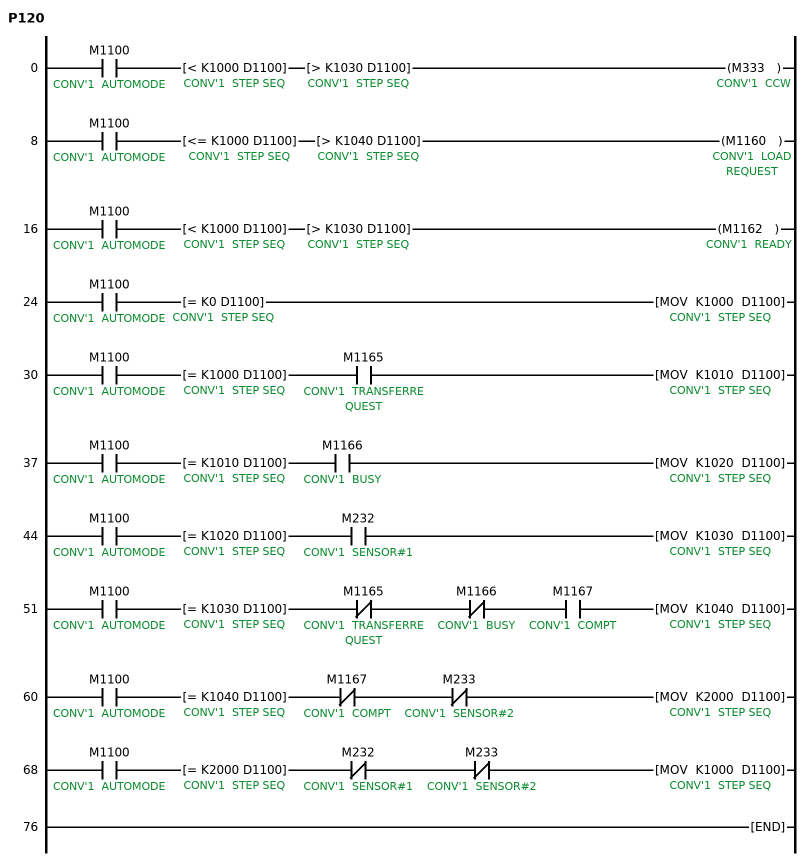
[picture p24: ladder of P120, rungs at steps 0 to 76]
0     LD      M1100  ; CONV'1  AUTOMODE
      AND<    K1000 D1100  ; CONV'1  STEP SEQ
      AND>    K1030 D1100  ; CONV'1  STEP SEQ
      OUT     M333  ; CONV'1  CCW
8     LD      M1100  ; CONV'1  AUTOMODE
      AND<=   K1000 D1100  ; CONV'1  STEP SEQ
      AND>    K1040 D1100  ; CONV'1  STEP SEQ
      OUT     M1160  ; CONV'1  LOAD    REQUEST
16    LD      M1100  ; CONV'1  AUTOMODE
      AND<    K1000 D1100  ; CONV'1  STEP SEQ
      AND>    K1030 D1100  ; CONV'1  STEP SEQ
      OUT     M1162  ; CONV'1  READY
24    LD      M1100  ; CONV'1  AUTOMODE
      AND=    K0 D1100  ; CONV'1  STEP SEQ
      MOV     K1000 D1100
30    LD      M1100  ; CONV'1  AUTOMODE
      AND=    K1000 D1100  ; CONV'1  STEP SEQ
      AND     M1165  ; CONV'1  TRANSFERREQUEST
      MOV     K1010 D1100
37    LD      M1100  ; CONV'1  AUTOMODE
      AND=    K1010 D1100  ; CONV'1  STEP SEQ
      AND     M1166  ; CONV'1  BUSY
      MOV     K1020 D1100
44    LD      M1100  ; CONV'1  AUTOMODE
      AND=    K1020 D1100  ; CONV'1  STEP SEQ
      AND     M232  ; CONV'1  SENSOR#1
      MOV     K1030 D1100
51    LD      M1100  ; CONV'1  AUTOMODE
      AND=    K1030 D1100  ; CONV'1  STEP SEQ
      ANI     M1165  ; CONV'1  TRANSFERREQUEST
      ANI     M1166  ; CONV'1  BUSY
      AND     M1167  ; CONV'1  COMPT
      MOV     K1040 D1100
60    LD      M1100  ; CONV'1  AUTOMODE
      AND=    K1040 D1100  ; CONV'1  STEP SEQ
      ANI     M1167  ; CONV'1  COMPT
      ANI     M233  ; CONV'1  SENSOR#2
      MOV     K2000 D1100
68    LD      M1100  ; CONV'1  AUTOMODE
      AND=    K2000 D1100  ; CONV'1  STEP SEQ
      ANI     M232  ; CONV'1  SENSOR#1
      ANI     M233  ; CONV'1  SENSOR#2
      MOV     K1000 D1100
76    END
END_PROGRAM

PROGRAM P130  // CONV2
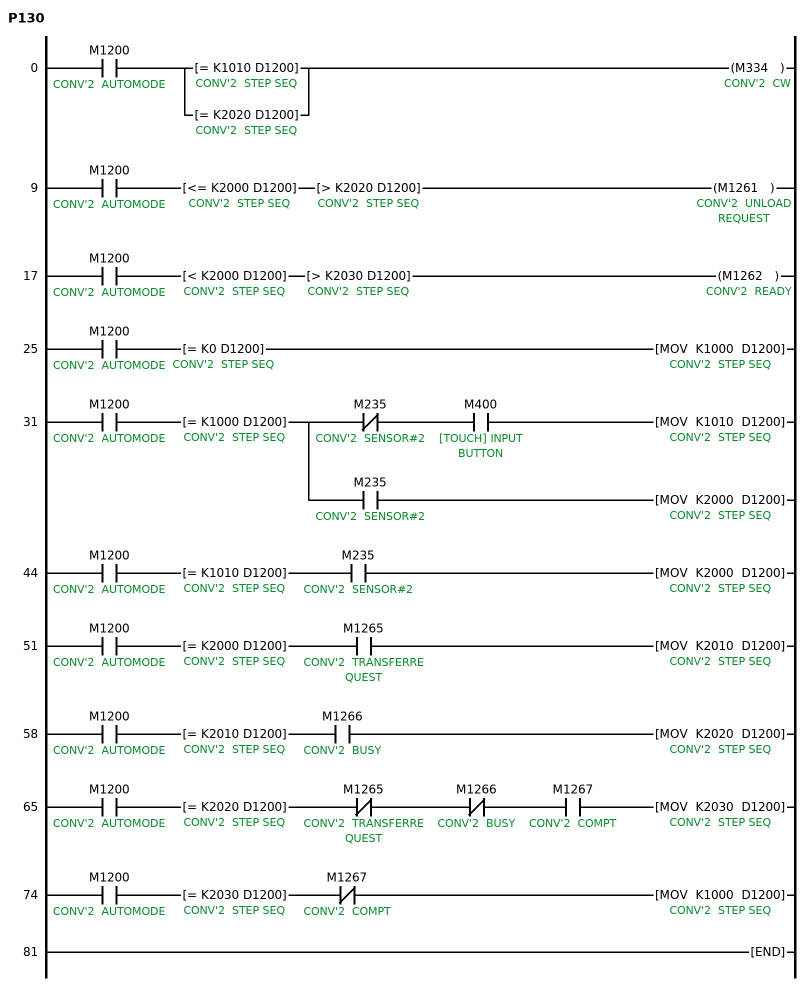
0     LD      M1200  ; CONV'2  AUTOMODE
      LD=     K1010 D1200  ; CONV'2  STEP SEQ
      OR=     K2020 D1200  ; CONV'2  STEP SEQ
      ANB
      OUT     M334  ; CONV'2  CW
9     LD      M1200  ; CONV'2  AUTOMODE
      AND<=   K2000 D1200  ; CONV'2  STEP SEQ
      AND>    K2020 D1200  ; CONV'2  STEP SEQ
      OUT     M1261  ; CONV'2  UNLOAD  REQUEST
17    LD      M1200  ; CONV'2  AUTOMODE
      AND<    K2000 D1200  ; CONV'2  STEP SEQ
      AND>    K2030 D1200  ; CONV'2  STEP SEQ
      OUT     M1262  ; CONV'2  READY
25    LD      M1200  ; CONV'2  AUTOMODE
      AND=    K0 D1200  ; CONV'2  STEP SEQ
      MOV     K1000 D1200
31    LD      M1200  ; CONV'2  AUTOMODE
      AND=    K1000 D1200  ; CONV'2  STEP SEQ
      MPS
      ANI     M235  ; CONV'2  SENSOR#2
      AND     M400  ; [TOUCH] INPUT   BUTTON
      MOV     K1010 D1200
      MPP
      AND     M235  ; CONV'2  SENSOR#2
      MOV     K2000 D1200
44    LD      M1200  ; CONV'2  AUTOMODE
      AND=    K1010 D1200  ; CONV'2  STEP SEQ
      AND     M235  ; CONV'2  SENSOR#2
      MOV     K2000 D1200
51    LD      M1200  ; CONV'2  AUTOMODE
      AND=    K2000 D1200  ; CONV'2  STEP SEQ
      AND     M1265  ; CONV'2  TRANSFERREQUEST
      MOV     K2010 D1200
58    LD      M1200  ; CONV'2  AUTOMODE
      AND=    K2010 D1200  ; CONV'2  STEP SEQ
      AND     M1266  ; CONV'2  BUSY
      MOV     K2020 D1200
65    LD      M1200  ; CONV'2  AUTOMODE
      AND=    K2020 D1200  ; CONV'2  STEP SEQ
      ANI     M1265  ; CONV'2  TRANSFERREQUEST
      ANI     M1266  ; CONV'2  BUSY
      AND     M1267  ; CONV'2  COMPT
      MOV     K2030 D1200
74    LD      M1200  ; CONV'2  AUTOMODE
      AND=    K2030 D1200  ; CONV'2  STEP SEQ
      ANI     M1267  ; CONV'2  COMPT
      MOV     K1000 D1200
81    END
END_PROGRAM

PROGRAM P140  // CONV3
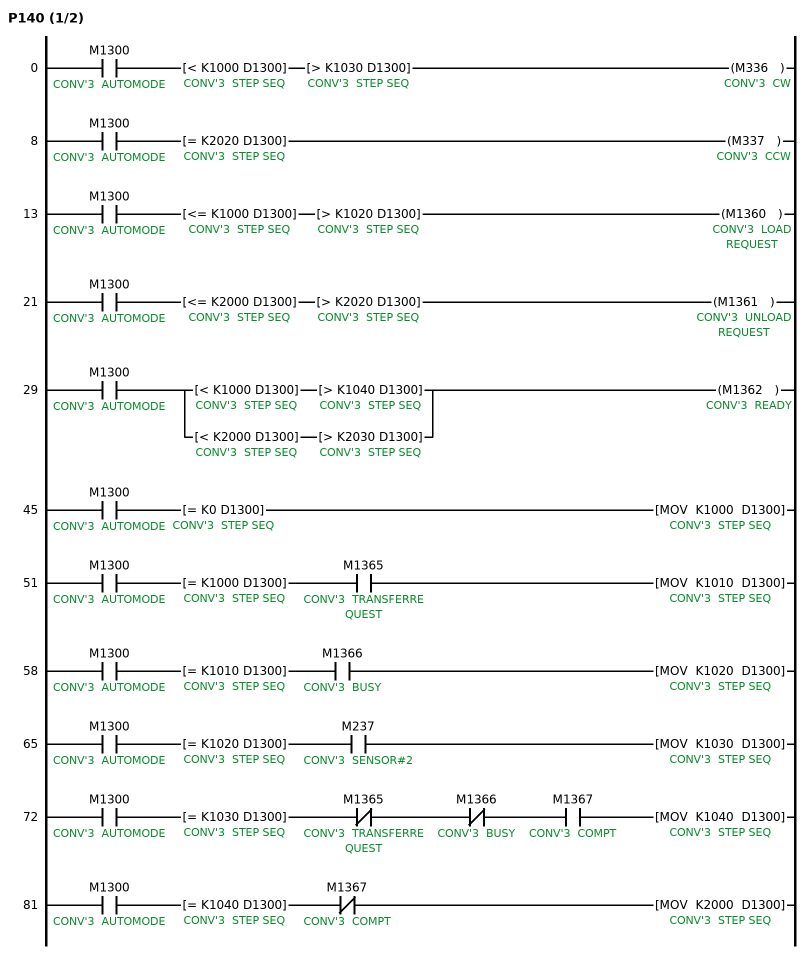
0     LD      M1300  ; CONV'3  AUTOMODE
      AND<    K1000 D1300  ; CONV'3  STEP SEQ
      AND>    K1030 D1300  ; CONV'3  STEP SEQ
      OUT     M336  ; CONV'3  CW
8     LD      M1300  ; CONV'3  AUTOMODE
      AND=    K2020 D1300  ; CONV'3  STEP SEQ
      OUT     M337  ; CONV'3  CCW
13    LD      M1300  ; CONV'3  AUTOMODE
      AND<=   K1000 D1300  ; CONV'3  STEP SEQ
      AND>    K1020 D1300  ; CONV'3  STEP SEQ
      OUT     M1360  ; CONV'3  LOAD    REQUEST
21    LD      M1300  ; CONV'3  AUTOMODE
      AND<=   K2000 D1300  ; CONV'3  STEP SEQ
      AND>    K2020 D1300  ; CONV'3  STEP SEQ
      OUT     M1361  ; CONV'3  UNLOAD  REQUEST
29    LD      M1300  ; CONV'3  AUTOMODE
      LD<     K1000 D1300  ; CONV'3  STEP SEQ
      AND>    K1040 D1300  ; CONV'3  STEP SEQ
      LD<     K2000 D1300  ; CONV'3  STEP SEQ
      AND>    K2030 D1300  ; CONV'3  STEP SEQ
      ORB
      ANB
      OUT     M1362  ; CONV'3  READY
45    LD      M1300  ; CONV'3  AUTOMODE
      AND=    K0 D1300  ; CONV'3  STEP SEQ
      MOV     K1000 D1300
51    LD      M1300  ; CONV'3  AUTOMODE
      AND=    K1000 D1300  ; CONV'3  STEP SEQ
      AND     M1365  ; CONV'3  TRANSFERREQUEST
      MOV     K1010 D1300
58    LD      M1300  ; CONV'3  AUTOMODE
      AND=    K1010 D1300  ; CONV'3  STEP SEQ
      AND     M1366  ; CONV'3  BUSY
      MOV     K1020 D1300
65    LD      M1300  ; CONV'3  AUTOMODE
      AND=    K1020 D1300  ; CONV'3  STEP SEQ
      AND     M237  ; CONV'3  SENSOR#2
      MOV     K1030 D1300
72    LD      M1300  ; CONV'3  AUTOMODE
      AND=    K1030 D1300  ; CONV'3  STEP SEQ
      ANI     M1365  ; CONV'3  TRANSFERREQUEST
      ANI     M1366  ; CONV'3  BUSY
      AND     M1367  ; CONV'3  COMPT
      MOV     K1040 D1300
81    LD      M1300  ; CONV'3  AUTOMODE
      AND=    K1040 D1300  ; CONV'3  STEP SEQ
      ANI     M1367  ; CONV'3  COMPT
      MOV     K2000 D1300
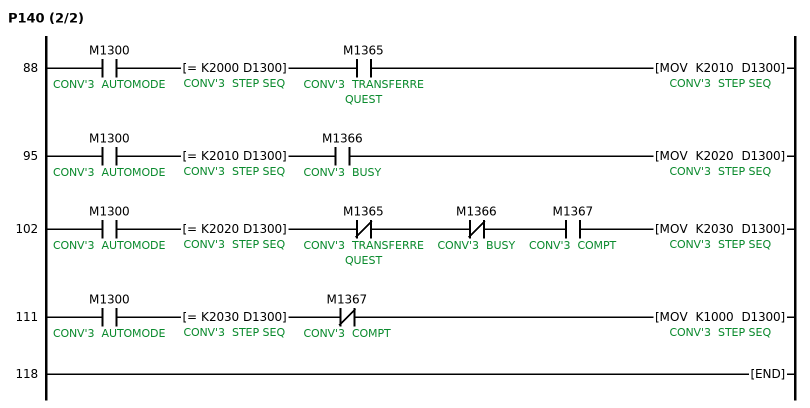
88    LD      M1300  ; CONV'3  AUTOMODE
      AND=    K2000 D1300  ; CONV'3  STEP SEQ
      AND     M1365  ; CONV'3  TRANSFERREQUEST
      MOV     K2010 D1300
95    LD      M1300  ; CONV'3  AUTOMODE
      AND=    K2010 D1300  ; CONV'3  STEP SEQ
      AND     M1366  ; CONV'3  BUSY
      MOV     K2020 D1300
102   LD      M1300  ; CONV'3  AUTOMODE
      AND=    K2020 D1300  ; CONV'3  STEP SEQ
      ANI     M1365  ; CONV'3  TRANSFERREQUEST
      ANI     M1366  ; CONV'3  BUSY
      AND     M1367  ; CONV'3  COMPT
      MOV     K2030 D1300
111   LD      M1300  ; CONV'3  AUTOMODE
      AND=    K2030 D1300  ; CONV'3  STEP SEQ
      ANI     M1367  ; CONV'3  COMPT
      MOV     K1000 D1300
118   END
END_PROGRAM

PROGRAM P150  // CONV4
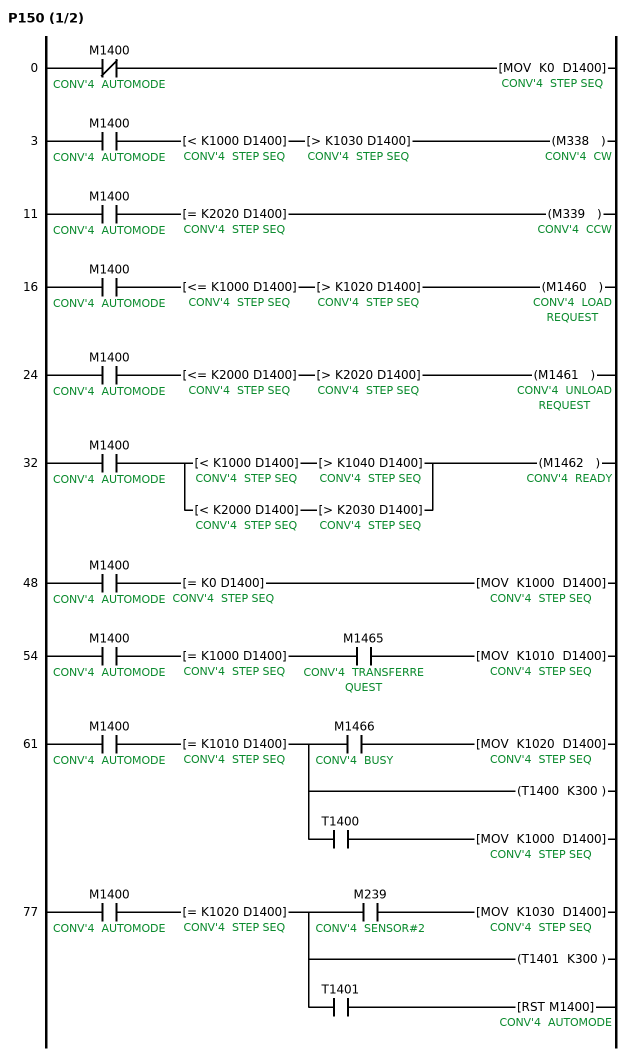
0     LDI     M1400  ; CONV'4  AUTOMODE
      MOV     K0 D1400  ; CONV'4  STEP SEQ
3     LD      M1400  ; CONV'4  AUTOMODE
      AND<    K1000 D1400  ; CONV'4  STEP SEQ
      AND>    K1030 D1400  ; CONV'4  STEP SEQ
      OUT     M338  ; CONV'4  CW
11    LD      M1400  ; CONV'4  AUTOMODE
      AND=    K2020 D1400  ; CONV'4  STEP SEQ
      OUT     M339  ; CONV'4  CCW
16    LD      M1400  ; CONV'4  AUTOMODE
      AND<=   K1000 D1400  ; CONV'4  STEP SEQ
      AND>    K1020 D1400  ; CONV'4  STEP SEQ
      OUT     M1460  ; CONV'4  LOAD    REQUEST
24    LD      M1400  ; CONV'4  AUTOMODE
      AND<=   K2000 D1400  ; CONV'4  STEP SEQ
      AND>    K2020 D1400  ; CONV'4  STEP SEQ
      OUT     M1461  ; CONV'4  UNLOAD  REQUEST
32    LD      M1400  ; CONV'4  AUTOMODE
      LD<     K1000 D1400  ; CONV'4  STEP SEQ
      AND>    K1040 D1400  ; CONV'4  STEP SEQ
      LD<     K2000 D1400  ; CONV'4  STEP SEQ
      AND>    K2030 D1400  ; CONV'4  STEP SEQ
      ORB
      ANB
      OUT     M1462  ; CONV'4  READY
48    LD      M1400  ; CONV'4  AUTOMODE
      AND=    K0 D1400  ; CONV'4  STEP SEQ
      MOV     K1000 D1400
54    LD      M1400  ; CONV'4  AUTOMODE
      AND=    K1000 D1400  ; CONV'4  STEP SEQ
      AND     M1465  ; CONV'4  TRANSFERREQUEST
      MOV     K1010 D1400
61    LD      M1400  ; CONV'4  AUTOMODE
      AND=    K1010 D1400  ; CONV'4  STEP SEQ
      MPS
      AND     M1466  ; CONV'4  BUSY
      MOV     K1020 D1400
      MPP
      OUT     T1400 K300
      AND     T1400
      MOV     K1000 D1400
77    LD      M1400  ; CONV'4  AUTOMODE
      AND=    K1020 D1400  ; CONV'4  STEP SEQ
      MPS
      AND     M239  ; CONV'4  SENSOR#2
      MOV     K1030 D1400
      MPP
      OUT     T1401 K300
      AND     T1401
      RST     M1400  ; CONV'4  AUTOMODE
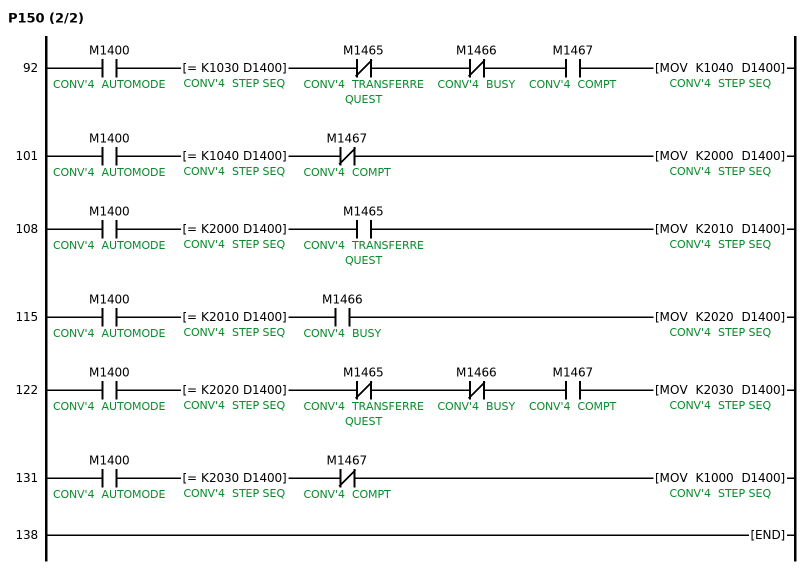
92    LD      M1400  ; CONV'4  AUTOMODE
      AND=    K1030 D1400  ; CONV'4  STEP SEQ
      ANI     M1465  ; CONV'4  TRANSFERREQUEST
      ANI     M1466  ; CONV'4  BUSY
      AND     M1467  ; CONV'4  COMPT
      MOV     K1040 D1400
101   LD      M1400  ; CONV'4  AUTOMODE
      AND=    K1040 D1400  ; CONV'4  STEP SEQ
      ANI     M1467  ; CONV'4  COMPT
      MOV     K2000 D1400
108   LD      M1400  ; CONV'4  AUTOMODE
      AND=    K2000 D1400  ; CONV'4  STEP SEQ
      AND     M1465  ; CONV'4  TRANSFERREQUEST
      MOV     K2010 D1400
115   LD      M1400  ; CONV'4  AUTOMODE
      AND=    K2010 D1400  ; CONV'4  STEP SEQ
      AND     M1466  ; CONV'4  BUSY
      MOV     K2020 D1400
122   LD      M1400  ; CONV'4  AUTOMODE
      AND=    K2020 D1400  ; CONV'4  STEP SEQ
      ANI     M1465  ; CONV'4  TRANSFERREQUEST
      ANI     M1466  ; CONV'4  BUSY
      AND     M1467  ; CONV'4  COMPT
      MOV     K2030 D1400
131   LD      M1400  ; CONV'4  AUTOMODE
      AND=    K2030 D1400  ; CONV'4  STEP SEQ
      ANI     M1467  ; CONV'4  COMPT
      MOV     K1000 D1400
138   END
END_PROGRAM

PROGRAM P100  // MODE
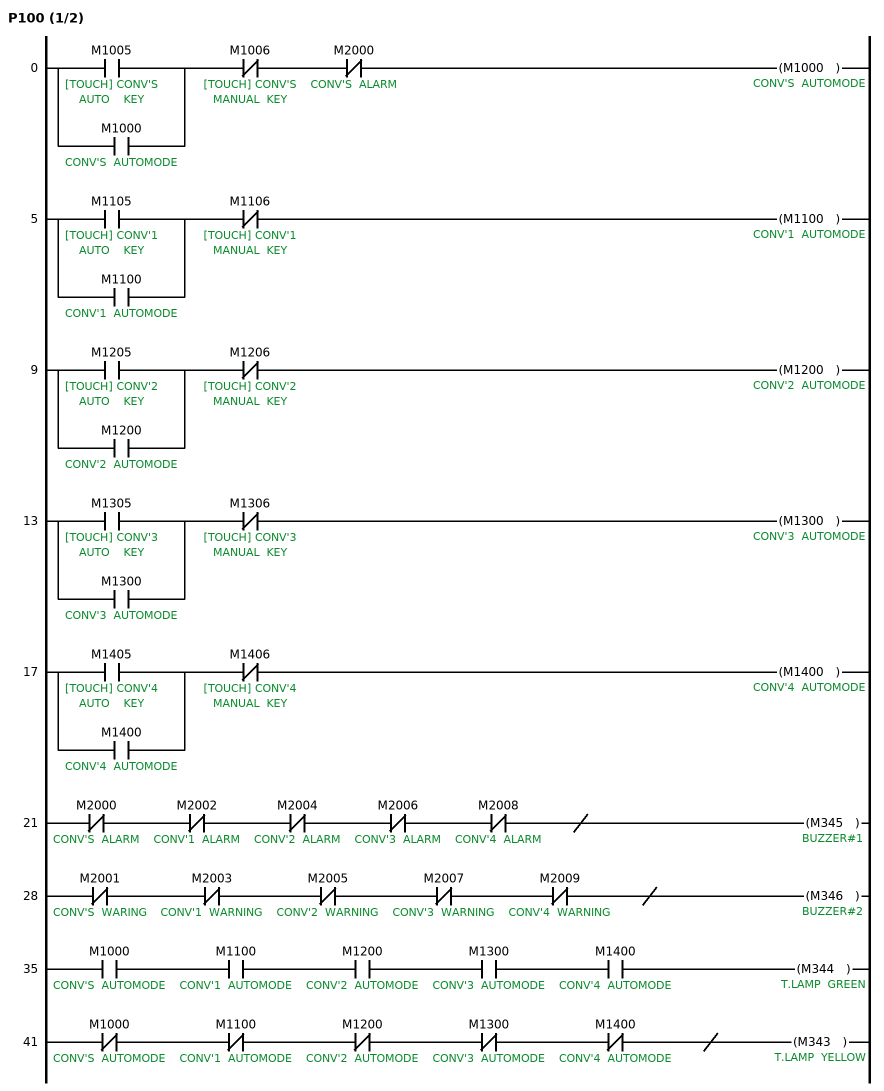
0     LD      M1005  ; [TOUCH] CONV'S  AUTO    KEY
      OR      M1000  ; CONV'S  AUTOMODE
      ANI     M1006  ; [TOUCH] CONV'S  MANUAL  KEY
      ANI     M2000  ; CONV'S  ALARM
      OUT     M1000  ; CONV'S  AUTOMODE
5     LD      M1105  ; [TOUCH] CONV'1  AUTO    KEY
      OR      M1100  ; CONV'1  AUTOMODE
      ANI     M1106  ; [TOUCH] CONV'1  MANUAL  KEY
      OUT     M1100  ; CONV'1  AUTOMODE
9     LD      M1205  ; [TOUCH] CONV'2  AUTO    KEY
      OR      M1200  ; CONV'2  AUTOMODE
      ANI     M1206  ; [TOUCH] CONV'2  MANUAL  KEY
      OUT     M1200  ; CONV'2  AUTOMODE
13    LD      M1305  ; [TOUCH] CONV'3  AUTO    KEY
      OR      M1300  ; CONV'3  AUTOMODE
      ANI     M1306  ; [TOUCH] CONV'3  MANUAL  KEY
      OUT     M1300  ; CONV'3  AUTOMODE
17    LD      M1405  ; [TOUCH] CONV'4  AUTO    KEY
      OR      M1400  ; CONV'4  AUTOMODE
      ANI     M1406  ; [TOUCH] CONV'4  MANUAL  KEY
      OUT     M1400  ; CONV'4  AUTOMODE
21    LDI     M2000  ; CONV'S  ALARM
      ANI     M2002  ; CONV'1  ALARM
      ANI     M2004  ; CONV'2  ALARM
      ANI     M2006  ; CONV'3  ALARM
      ANI     M2008  ; CONV'4  ALARM
      INV
      OUT     M345  ; BUZZER#1
28    LDI     M2001  ; CONV'S  WARING
      ANI     M2003  ; CONV'1  WARNING
      ANI     M2005  ; CONV'2  WARNING
      ANI     M2007  ; CONV'3  WARNING
      ANI     M2009  ; CONV'4  WARNING
      INV
      OUT     M346  ; BUZZER#2
35    LD      M1000  ; CONV'S  AUTOMODE
      AND     M1100  ; CONV'1  AUTOMODE
      AND     M1200  ; CONV'2  AUTOMODE
      AND     M1300  ; CONV'3  AUTOMODE
      AND     M1400  ; CONV'4  AUTOMODE
      OUT     M344  ; T.LAMP  GREEN
41    LDI     M1000  ; CONV'S  AUTOMODE
      ANI     M1100  ; CONV'1  AUTOMODE
      ANI     M1200  ; CONV'2  AUTOMODE
      ANI     M1300  ; CONV'3  AUTOMODE
      ANI     M1400  ; CONV'4  AUTOMODE
      INV
      OUT     M343  ; T.LAMP  YELLOW
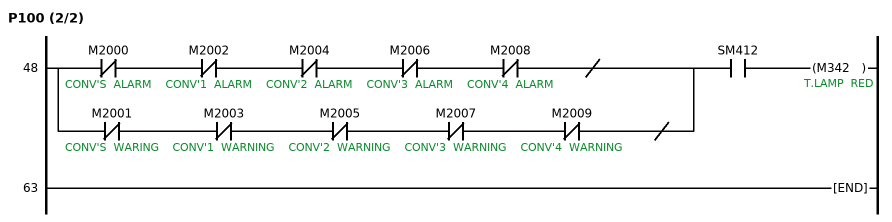
48    LDI     M2000  ; CONV'S  ALARM
      ANI     M2002  ; CONV'1  ALARM
      ANI     M2004  ; CONV'2  ALARM
      ANI     M2006  ; CONV'3  ALARM
      ANI     M2008  ; CONV'4  ALARM
      INV
      LDI     M2001  ; CONV'S  WARING
      ANI     M2003  ; CONV'1  WARNING
      ANI     M2005  ; CONV'2  WARNING
      ANI     M2007  ; CONV'3  WARNING
      ANI     M2009  ; CONV'4  WARNING
      INV
      ORB
      AND     SM412
      OUT     M342  ; T.LAMP  RED
63    END
END_PROGRAM

// device comments not shown above
M1060  ; CONV    2 -> S  READY
M1061  ; CONV    2 -> S  BUSY
M1070  ; CONV    S -> 1  READY
M1071  ; CONV    S -> 1  BUSY
M1110  ; CONV'1  CW
M1111  ; CONV'1  CW
M1115  ; CONV'1  CCW
M1116  ; CONV'1  CCW
M1210  ; CONV'2  CW
M1211  ; CONV'2  CW
